	MaxKO_OLD		: REAL;
	i 				: INT;
END_VAR

RT_CLK_A(CLK:= CLK_A);
RT_CLK_B(CLK:= CLK_B);
RT_CLK_Forming(CLK:= CLK_Forming);

IF init THEN
	i := 1;
	WHILE i <= 6 DO
		MaxKO_Array[i] := 0;
		i := i +1;
	END_WHILE
	MaxKO := 0;
END_IF

IF RT_CLK_A.Q THEN
	CLK_A := FALSE;
	MaxKO_Array[2] := MaxKO_Array[1];
	MaxKO_Array[1] := Value_A;
	IF NOT BEnabled THEN
		MaxKO_Array[4] := MaxKO_Array[3];
		MaxKO_Array[3] := Value_A;
	END_IF
END_IF
IF RT_CLK_B.Q THEN
	CLK_B := FALSE;
	MaxKO_Array[4] := MaxKO_Array[3];
	MaxKO_Array[3] := Value_B;
	IF NOT AEnabled THEN
		MaxKO_Array[2] := MaxKO_Array[1];
		MaxKO_Array[1] := Value_B;
	END_IF
END_IF
IF RT_CLK_Forming.Q THEN
	CLK_Forming := FALSE;
	MaxKO_Array[6] := MaxKO_Array[5];
	MaxKO_Array[5] := Value_Forming;
END_IF

IF RT_CLK_A.Q OR RT_CLK_B.Q OR RT_CLK_Forming.Q  THEN
	(*i := 1;
	WHILE i <= 5 DO
		IF MaxKO_Array[i] > MaxKO_Array[i+1] THEN
			MaxKO := MaxKO_Array[i+1];
		ELSIF MaxKO_Array[i+1] < MaxKO_OLD THEN
			MaxKO := MaxKO_Array[i];
		ELSE
			MaxKO := MaxKO_OLD;
		END_IF
		MaxKO_OLD := MaxKo;
		i := i+1;
	END_WHILE*)
	
	MaxKO := MIN(MIN(MIN(MIN(MIN(MaxKO_Array[1],MaxKO_Array[2]),MaxKO_Array[3]),MaxKO_Array[4]),MaxKO_Array[5]),MaxKO_Array[6]);
END_IF

END_FUNCTION_BLOCK

// ---- POUs/Standard/HydraulicCylinderAnalog/FB_HydraulicCilinderAnalog_.TcPOU
FUNCTION_BLOCK FB_HydraulicCilinderAnalog_

VAR_INPUT

	mxReset							: BOOL;	(*Reset Error*)
	mxEmergency						: BOOL;
	mxAutoMode						: BOOL; (* TRUE = Automode *)
	EndPositionIn					: REAL;
	EndPositionOut					: REAL;
	OffsetPosition					: REAL;
	OffsetAlarmPosition				: REAL;	
	PositionPhysicalMeasured		: REAL;	
	RHSR_Blocked					: BOOL; (*IF true, then movement of the cylinder is blocked by the red hot safetyrules.*)
	
	ManSpeedCreepIn					: REAL;
	ManSpeedCreepOut				: REAL;
	ManSpeedSlowIn					: REAL;
	ManSpeedSlowOut					: REAL;
	ManSpeedIn						: REAL;
	ManSpeedOut						: REAL;

END_VAR
VAR_OUTPUT
(*Errors*)
	Errors							: ST_HydraulicErrorsAnalog;
	mxErrorInit						: BOOL;		(* Error, stop immediately. Initialisation neccesary *)
	mxErrorStopinPos				: BOOL;		(* Error, stop in position. Only reset neccesary *)

(* State vars *)
	mxCycleBusy						: BOOL;
	mxInitBusy						: BOOL;
	
(* Vars *)
	mxInitialized					: BOOL;
	ActPosition						: REAL;
	ActMeasuredPosition				: REAL;
	mxSlowActive					: BOOL;
	mxIsMovingIn					: BOOL;
	mxIsMovingOut					: BOOL;
	mxIsIn							: BOOL;
	mxIsOut							: BOOL;
	mxMoveIn						: BOOL;
	mxMoveOut						: BOOL;
END_VAR
VAR
	RodSidePressure					: FB_AnalogIn4_20mA;
	BottomSidePressure				: FB_AnalogIn4_20mA;

	(* Objects *)
	HydraulicValve					: FB_AnalogOutMinus10_10V;
	HydraulicPos 					: FB_BalluffPosition;
	MachPar							: ST_HydraulicCilinderMachParAnalog;
	
	EndPosition						: REAL; (* Destination position *)
	SlowPosition					: REAL; (* Slow position *)

	FT_ValveInOff					: F_TRIG;
	FT_ValveOutOff					: F_TRIG;
	HydraulicStoredPosition			: REAL;
	
	ixEndSwitchA					AT %I* : BOOL;
	ixEndSwitchB					AT %I* : BOOL;
	ixMSPAReadyToOperate			AT %I* : BOOL;
	qxMSPAEnable					AT %Q* : BOOL;
	
	mxMoveReadyWithoutMoving		: BOOL;
	
	RT_Emergency: R_Trig;
	FT_AutoMode: F_TRIG;
	SafePosReached: BOOL;
	Mancreep: BOOL;
	ManCreepUp: BOOL;
	ManSlowUp: BOOL;
	ManUp: BOOL;
	ManCreepDown: BOOL;
	ManSlowDown: BOOL;
	ManDown: BOOL;
	SR_RodSidePressureTooHigh: SR;
	SR_BotSidePressureTooHigh: SR;
	T_EmergencyDelay: TON;
	RT_EmergencyDelay: R_TRIG;
	T_EnableDelayedOff: TOF;
	mxTestValue: REAL;
	FT_ValveToNeutralPos: F_trig;
	SR_SafePositionNotReached: SR;
END_VAR
VAR_IN_OUT
	PositionPhysicalMeasuredOld		: REAL;
	PhysicalOffsetPos				: REAL;
END_VAR

Error();
Objects();
Manual();

RT_Emergency(CLK:= mxEmergency);
FT_AutoMode(CLK:=mxAutoMode);

// Enable MSPA2
T_EnableDelayedOff(IN:= NOT mxEmergency, PT:=T#500MS);
qxMSPAEnable := T_EnableDelayedOff.Q; 

// Calculate correction on actual balluf position to a virtual "zero" position.
IF PositionPhysicalMeasured <> PositionPhysicalMeasuredOld THEN
	PhysicalOffsetPos := (HydraulicPos.Position- (OffsetPosition + PositionPhysicalMeasured));
END_IF

// Create a virtual zero position by substracting a calculated offset
ActPosition:= HydraulicPos.Position - PhysicalOffsetPos;
ActMeasuredPosition:= HydraulicPos.Position;

mxIsMovingIn:= HydraulicValve.EngInput > 0;
mxIsMovingOut:= HydraulicValve.EngInput < 0;

// Hysteresis + 2 to enlarge the RHSR window.
mxIsIn:= (ActPosition <= (EndPositionIn + (MachPar.Hysteresis + 2))) AND (ActPosition >= (EndPositionIn - (MachPar.Hysteresis + 2)));
mxIsOut:= (ActPosition <= (EndPositionOut + (MachPar.Hysteresis + 2))) AND (ActPosition >= (EndPositionOut - (MachPar.Hysteresis + 2)));

(*Overwrite previous value*)
PositionPhysicalMeasuredOld := PositionPhysicalMeasured;

// Close valves on emergency stop.
IF RT_Emergency.Q OR FT_AutoMode.Q THEN
	HydraulicValve.EngInput := 0;
END_IF

// From the TOP bosch -> If both feedback signals are high, the valve can be considered "safe" (base position reached
SafePosReached:= ixEndSwitchA AND ixEndSwitchB;

ACTION Error:
Errors.BallufError:= HydraulicPos.Error;

// Check for a to high a pressure
SR_RodSidePressureTooHigh(SET1:=mxIsMovingIn AND (RodSidePressure.EngFilt > MachPar.MaxRodSidePressure),Reset:=mxReset,Q1=>Errors.RodSidePressureTooHigh);
SR_BotSidePressureTooHigh(SET1:=mxIsMovingOut AND (BottomSidePressure.EngFilt > MachPar.MaxBotSidePressure),Reset:=mxReset,Q1=>Errors.BotSidePressureTooHigh);	 

SR_SafePositionNotReached(SET1:=T_EmergencyDelay.Q AND NOT SafePosReached, reset:=mxReset, Q1=>Errors.SafePositionValveNotReached);

// Delay the emstop from the doors open, and wait checking on position.
T_EmergencyDelay(IN:=mxEmergency, PT:=T#500MS);
RT_EmergencyDelay(CLK:=T_EmergencyDelay.Q);

(* Als valve up/down uit gaat, positie opslaan en controleren of deze veranderd tov de act positie*)
IF RT_EmergencyDelay.Q THEN 
	HydraulicStoredPosition:= ActPosition; 
END_IF
IF mxReset THEN
	HydraulicStoredPosition:= ActPosition;
	Errors.IsMovingWithoutActivation:= FALSE;
ELSIF (T_EmergencyDelay.Q OR (HydraulicValve.EngInput = 0)) AND ((HydraulicStoredPosition > (ActPosition + 10)) OR (HydraulicStoredPosition < (ActPosition - 10))) THEN
	//Errors.IsMovingWithoutActivation:= TRUE;
END_IF

// Look into above alarm, this keeps triggering, probably due to not setting actual position in the right way

(***************************************************************************************)
mxErrorStopInPos:= FALSE;
mxErrorInit:= Errors.IsMovingWithoutActivation; //OR Errors.BotSidePressureTooHigh OR Errors.RodSidePressureTooHigh;
END_ACTION

METHOD M_Move : BOOL
VAR_INPUT
	EndPosition		: REAL; (* Destination position *)
	NormalSpeed		: REAL;
	
	SlowPosition	: REAL; (* Slow position *)
	SlowSpeed		: REAL;
		
	CreepPosition 	: REAL;	(*CreepSpeed.*)
	CreepSpeed		: REAL;
	
END_VAR
VAR_OUTPUT
END_VAR
VAR


	mxMoveINReady: BOOL;
	mxMoveOutReady: BOOL;
	ActSpeed : real;
END_VAR
mxMoveReadyWithoutMoving := FALSE;

//Check current position of the rod, and check where to go and detemine direction
IF ActPosition > (EndPosition + MachPar.Hysteresis) THEN		// Move up (Positive)
	(*Set movement direction bit.*)
	mxMoveIn:= FALSE;
	mxMoveOut:= TRUE;
	ActSpeed:= NormalSpeed;
ELSIF ActPosition < (EndPosition - MachPar.Hysteresis) THEN 	// Move Down (Negative)
	(*Set movement direction bit.*)
	mxMoveIn:= TRUE;
	mxMoveOut:= FALSE;
	ActSpeed:= NormalSpeed;
ELSE																			// Don't move at all (allready on pos).
	mxMoveIn:= FALSE;
	mxMoveOut:= FALSE;
	mxMoveReadyWithoutMoving := TRUE;
END_IF

// Check at which speed the movement needs to be done.
IF (NOT mxMoveIn AND NOT mxMoveOut) THEN	// No movement.
	ActSpeed:= 0;
ELSIF (mxMoveIn AND (ActPosition > CreepPosition)) OR (mxMoveOut AND (ActPosition < CreepPosition)) THEN 	//Creep speed.
	ActSpeed:= CreepSpeed;
ELSIF (mxMoveIn AND (ActPosition > SlowPosition)) OR (mxMoveOut AND (ActPosition < SlowPosition)) THEN 		//Slow speed.
	ActSpeed:= SlowSpeed;
ELSIF (mxMoveIn OR mxMoveOut) THEN	// Normal speed if nothing else is selected.
	ActSpeed:= NormalSpeed;
END_IF

// Set actual output on valve.
IF mxMoveOut THEN ActSpeed := Actspeed *-1; END_IF
HydraulicValve.EngInput := ActSpeed;

// Check if the movement is ready.
mxMoveInReady := (mxMoveIn AND ((ActPosition >= (EndPosition - MachPar.Hysteresis)) AND 
				(ActPosition <= (EndPosition + MachPar.Hysteresis))));
mxMoveOutReady := (mxMoveOut AND ((ActPosition >= (EndPosition - MachPar.Hysteresis)) AND 
				(ActPosition <= (EndPosition + MachPar.Hysteresis))));	

// reset directional bits to zero when leaving this method.
IF mxMoveInReady OR mxMoveOutReady OR mxMoveReadyWithoutMoving THEN
	mxMoveIn:= FALSE;
	mxMoveOut:= FALSE;
END_IF

// Signal the method has finished to the caller of the method.
M_MOVE := mxMoveInReady OR mxMoveOutReady OR mxMoveReadyWithoutMoving;
END_METHOD

METHOD M_OpenAndMove : BOOL
VAR_INPUT
	EndPosition		: REAL; (* Destination position *)
	NormalSpeed		: REAL;
	
	SlowPosition	: REAL; (* Slow position *)
	SlowSpeed		: REAL;
		
	CreepPosition 	: REAL;	(*CreepSpeed.*)
	CreepSpeed		: REAL;
	
	OpenPosition	: REAL;
	OpenSpeed		: REAL;
	
END_VAR
VAR_OUTPUT
END_VAR
VAR


	mxMoveINReady: BOOL;
	mxMoveOutReady: BOOL;
	ActSpeed : real;
END_VAR
mxMoveReadyWithoutMoving := FALSE;

//Check current position of the rod, and check where to go and detemine direction
IF ActPosition > (EndPosition + MachPar.Hysteresis) THEN		// Move up (Positive)
	(*Set movement direction bit.*)
	mxMoveIn:= FALSE;
	mxMoveOut:= TRUE;
	ActSpeed:= NormalSpeed;
ELSIF ActPosition < (EndPosition - MachPar.Hysteresis) THEN 	// Move Down (Negative)
	(*Set movement direction bit.*)
	mxMoveIn:= TRUE;
	mxMoveOut:= FALSE;
	ActSpeed:= NormalSpeed;
ELSE																			// Don't move at all (allready on pos).
	mxMoveIn:= FALSE;
	mxMoveOut:= FALSE;
	mxMoveReadyWithoutMoving := TRUE;
END_IF

// Check at which speed the movement needs to be done.
IF (NOT mxMoveIn AND NOT mxMoveOut) THEN	// No movement.
	ActSpeed:= 0;
ELSIF (mxMoveIn AND (ActPosition > CreepPosition)) OR (mxMoveOut AND (ActPosition < CreepPosition)) THEN 	//Creep speed.
	ActSpeed:= CreepSpeed;
ELSIF (mxMoveIn AND (ActPosition > SlowPosition)) OR (mxMoveOut AND (ActPosition < SlowPosition)) THEN 		//Slow speed.
	ActSpeed:= SlowSpeed;
ELSIF (mxMoveIn AND (ActPosition < OpenPosition)) THEN 		//Only do this on way up.
	ActSpeed:= OpenSpeed;
ELSIF (mxMoveIn OR mxMoveOut) THEN	// Normal speed if nothing else is selected.
	ActSpeed:= NormalSpeed;
END_IF

// Set actual output on valve.
IF mxMoveOut THEN ActSpeed := Actspeed *-1; END_IF
HydraulicValve.EngInput := ActSpeed;

// Check if the movement is ready.
mxMoveInReady := (mxMoveIn AND ((ActPosition >= (EndPosition - MachPar.Hysteresis)) AND 
				(ActPosition <= (EndPosition + MachPar.Hysteresis))));
mxMoveOutReady := (mxMoveOut AND ((ActPosition >= (EndPosition - MachPar.Hysteresis)) AND 
				(ActPosition <= (EndPosition + MachPar.Hysteresis))));	

// reset directional bits to zero when leaving this method.
IF mxMoveInReady OR mxMoveOutReady OR mxMoveReadyWithoutMoving THEN
	mxMoveIn:= FALSE;
	mxMoveOut:= FALSE;
END_IF

// Signal the method has finished to the caller of the method.
M_OpenAndMove := mxMoveInReady OR mxMoveOutReady OR mxMoveReadyWithoutMoving;
END_METHOD

METHOD M_Press : BOOL
VAR_INPUT
	PressDown		 	: BOOL; // Determines if press needs to be done moving down 
	PressSpeed			: REAL;	// Flow at which the pressing occures
	StoppingPressure	: REAL;	// Pressure at which the pressing stops
END_VAR
VAR_OUTPUT
END_VAR
VAR
	PressingDone		: Bool;
END_VAR
IF PressDown THEN	// PressDown
	IF (BottomSidePressure.EngFilt < StoppingPressure - 15) THEN
		HydraulicValve.EngInput := PressSpeed * -1;
	END_IF
		
	IF (BottomSidePressure.EngFilt > StoppingPressure) THEN 
		HydraulicValve.EngInput := 0;			
		M_Press := TRUE;	// Signal the method is done.
	END_IF 	
ELSE				// PressUp
	IF (RodSidePressure.EngFilt < StoppingPressure) THEN
		HydraulicValve.EngInput := PressSpeed;
	ELSE
		HydraulicValve.EngInput := 0;	
		M_Press := TRUE;	// Signal the method is done.
	END_IF 
END_IF
END_METHOD

METHOD M_Stop : BOOL;
mxMoveIn := FALSE;
mxMoveOut := FALSE;

HydraulicValve.EngInput := 0.0;

M_Stop:= TRUE;
END_METHOD

METHOD M_StopDirect
HydraulicValve.EngInput := 0.0;
END_METHOD

ACTION Manual:
IF ManCreepUp THEN
	HydraulicValve.EngInput := ManSpeedCreepIn;
ELSIF ManSlowUp THEN
	HydraulicValve.EngInput := ManSpeedSlowIn;
ELSIF ManUp THEN
	HydraulicValve.EngInput := ManSpeedIn;
ELSIF ManCreepDown THEN
	HydraulicValve.EngInput := ManSpeedCreepOut * -1;
ELSIF ManSlowDown THEN
	HydraulicValve.EngInput := ManSpeedslowOut * -1;
ELSIF ManDown THEN											// Somebody is seriously wounded. ^_^
	HydraulicValve.EngInput := ManSpeedOut * -1;
END_IF

(*
FT_ValveToNeutralPos(CLK:=ManCreepUp OR ManSlowUp OR ManUp OR ManCreepDown OR ManSlowDown OR ManDown);

// When Automode is disabled, set the valve back to neutral position.
IF FT_AutoMode.Q OR Ft_ValveToNeutralPos.Q THEN
	HydraulicValve.EngInput := 0.0;
END_IF
*)
END_ACTION

ACTION Objects:
(* Objects Call *)
BottomSidePressure(
	EngLowLimit:=0, 
	EngUpperLimit:=315, 
	maOut=> , 
	EngUnits=> , 
	EngFilt=> , 
	OverRange=> , 
	UnderRange=> );

RodSidePressure(
	EngLowLimit:=0, 
	EngUpperLimit:=315, 
	maOut=> , 
	EngUnits=> , 
	EngFilt=> ,
	OverRange=> ,
	UnderRange=> );
	
HydraulicValve( 
	EngMin:= -100,
	EngMax:= 100,
	RHSR_Blocked:= RHSR_Blocked,
	VOut=> , 
	RawOut=> );
	
HydraulicPos();
END_ACTION

END_FUNCTION_BLOCK
